(* Logix 5000 project; controller BTS01 vendor 1 type 14 code 217 rev 32.14; software revision 32.04 *)

TASK MainTask (continuous, watchdog 500 ms) : MainProgram, Alarm, CIP

MODULES
   Local : vendor 1 type 14 code 217 (5069 0, rev 32.14)
      Flow_Meter_01 : Promag_300_500 (Ethernet 10.10.1.3, rev 1.1, StandardDataDriven RPI 20 ms)
      FLEX5000 : 5094-AENTR (Ethernet 10.10.1.2, rev 4.1)
          : 5094-IF8 (5094 1, rev 2.1, StandardDataDriven RPI 100 ms)
          : 5094-OB16 (5094 5, rev 2.1, StandardDataDriven RPI 5 ms)
              FLEX5000:5:O.Pt09.Data   // RED STOP
              FLEX5000:5:O.Pt08.Data   // GREEN RUN
          : 5094-IB16 (5094 3, rev 2.1, StandardDataDriven RPI 5 ms)
          : 5094-IB16 (5094 6, rev 2.1, StandardDataDriven RPI 5 ms)
          : 5094-OF8 (5094 2, rev 2.1, StandardDataDriven RPI 100 ms)
          : 5094-OB16 (5094 4, rev 2.1, StandardDataDriven RPI 5 ms)
              FLEX5000:4:O.Pt13.Data   // Red
END_MODULES

TYPE CIP_PROGRAM :   // 30 STEP CIP PROGRAM
STRUCT
   NAME : STRING;   // CIP PROGRAM NAME
   NUMBER : INT;   // CIP PROGRAM NUMBER
   STEPS : CIP_STEP_DEF[50];   // CIP PROGRAM STEPS
END_STRUCT
END_TYPE

TYPE CIP_Recipe :
STRUCT
   Recipe_Name : STRING;
   Recipe_Description : STRING;
   Step_Desc : STRING[50];
   Step_Time : REAL[50];
END_STRUCT
END_TYPE

TYPE CIP_STEP_DEF :   // CIP SEQUENCER STEP DEFFINITION
STRUCT
   NAME : STRING;   // CIP STEP NAME
   TYPE : INT;   // CIP STEP TYPE
   TIME_SPT : REAL;   // CIP STEP TIME
   RETURN_TEMP_SPT : REAL;   // CIP RETURN STEP TEMP
   REF_FILE : DINT;   // CIP STEP REFERENCE FILE
   RETURN_COND_SPT : REAL;   // CIP RETURN STEP CONDUCTIVITY
END_STRUCT
END_TYPE

TYPE DateTime :
STRUCT
   Year : DINT;
   Month : DINT;
   Day : DINT;
   Hour : DINT;
   Minute : DINT;
   Second : DINT;
   MicroSecond : DINT;
END_STRUCT
END_TYPE

TYPE STRING64 :
STRUCT
   LEN : DINT;
   DATA : SINT[64];
END_STRUCT
END_TYPE

ADD_ON_INSTRUCTION DTE_Air_Valve_v2   (* revision 2.0 *)
VAR_INPUT
   CMD : BOOL; {visible}
END_VAR
VAR_OUTPUT
   TON_OUT_ACC : DINT; {access Read Only, visible}
   TOFF_OUT_ACC : DINT; {access Read Only, visible}
   OUT : BOOL; {access Read Only, required}
END_VAR
VAR_INPUT
   FB_DES : BOOL;
   FB_ACT : BOOL;
   ACK : BOOL;
END_VAR
VAR_OUTPUT
   ALARME : BOOL; {access Read Only}
END_VAR
VAR_INPUT
   ALM_PRE : DINT := 7000;
   ALM_AUTO_RESET_PRE : DINT;
   TON_OUT_PRE : DINT; {required}
   TOFF_OUT_PRE : DINT; {required}
   P : BOOL; {required}   // Process Command
   C : BOOL; {required}   // CIP Command
   M : DINT;
        .1   // Auto On
        .2   // Force On
        .3   // Force Off
   desc_nom : DINT;
   equip_nom : DINT;
   nom : DINT;
   Allowed : BOOL;
END_VAR
VAR_IN_OUT
   Description : STRING; {required}
   PIDName : STRING; {required}
END_VAR
VAR_INPUT
   Auto_On_PB : BOOL; {required}   // Momentary PB
   Manual_On_PB : BOOL; {required}   // Momentary PB
   Manual_Off_PB : BOOL; {required}   // Momentary PB
   Status : DINT; {visible}
END_VAR
VAR_OUTPUT
   ITEMTAG : DINT; {access Read Only, visible}
END_VAR
VAR_INPUT
   MOA_Mode : DINT; {visible}
END_VAR
VAR
   INTERNAL_TIM_ALM : TIMER := (PRE := 7000);
   INTERNAL_TIM_AUTO_RESET : TIMER;
   OUT_OFF_MEM : BOOL;
   OUT_ON_MEM : BOOL;
   INTERNAL_TON_OUT : TIMER;
   INTERNAL_TOFF_OUT : TIMER;
   Desc : STRING;
   ValveName : STRING; {access None}
   DisplayName : STRING;
END_VAR

ROUTINE Logic   (* ladder *)
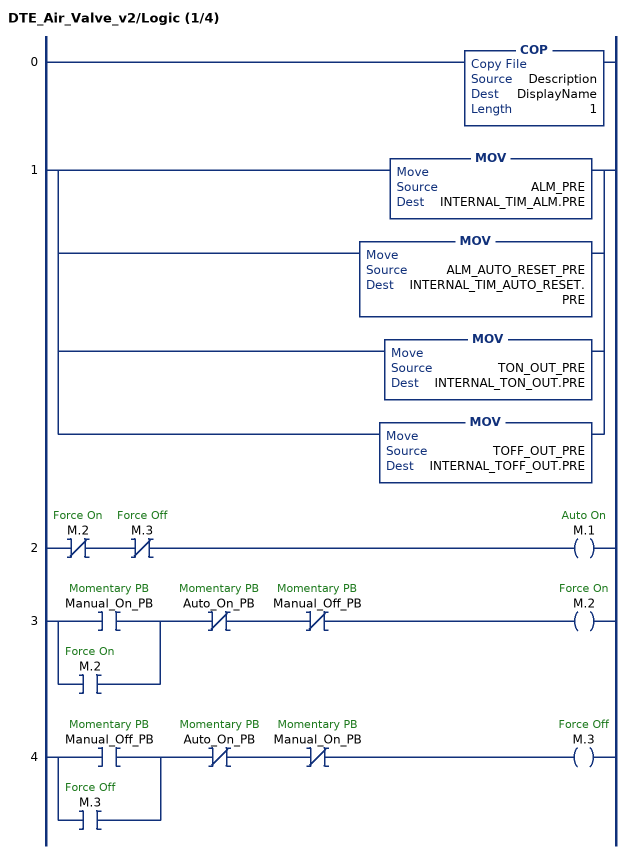
   0: COP(Description,DisplayName,1);
   1: [MOV(ALM_PRE,INTERNAL_TIM_ALM.PRE) ,MOV(ALM_AUTO_RESET_PRE,INTERNAL_TIM_AUTO_RESET.PRE) ,MOV(TON_OUT_PRE,INTERNAL_TON_OUT.PRE) ,MOV(TOFF_OUT_PRE,INTERNAL_TOFF_OUT.PRE) ];
   2: XIO(M.2)XIO(M.3)OTE(M.1);
   3: [XIC(Manual_On_PB) ,XIC(M.2) ]XIO(Auto_On_PB)XIO(Manual_Off_PB)OTE(M.2);
   4: [XIC(Manual_Off_PB) ,XIC(M.3) ]XIO(Auto_On_PB)XIO(Manual_On_PB)OTE(M.3);
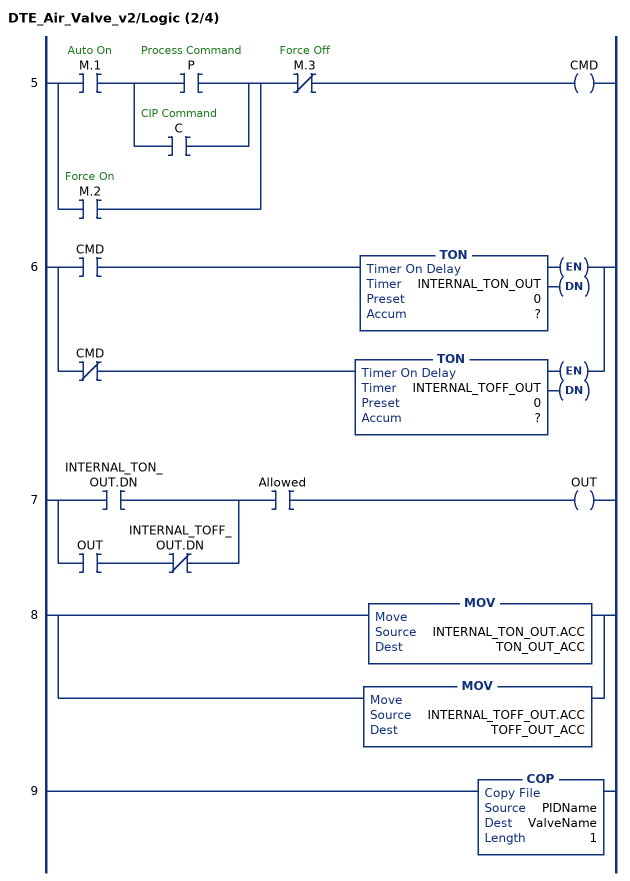
   5: [XIC(M.1) [XIC(P) ,XIC(C) ] ,XIC(M.2) ]XIO(M.3)OTE(CMD);
   6: [XIC(CMD) TON(INTERNAL_TON_OUT,?,?) ,XIO(CMD) TON(INTERNAL_TOFF_OUT,?,?) ];
   7: [XIC(INTERNAL_TON_OUT.DN) ,XIC(OUT) XIO(INTERNAL_TOFF_OUT.DN) ]XIC(Allowed)OTE(OUT);
   8: [MOV(INTERNAL_TON_OUT.ACC,TON_OUT_ACC) ,MOV(INTERNAL_TOFF_OUT.ACC,TOFF_OUT_ACC) ];
   9: COP(PIDName,ValveName,1);
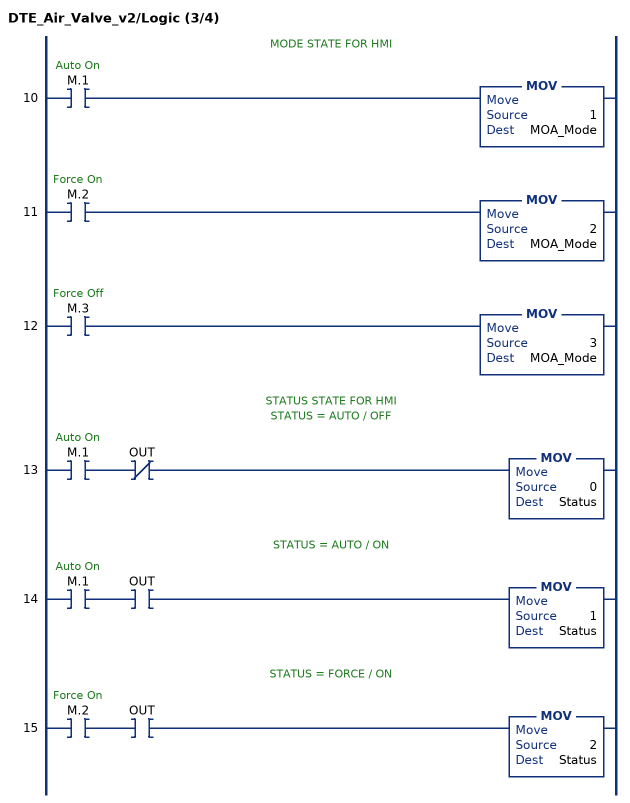
   // MODE STATE FOR HMI
   10: XIC(M.1)MOV(1,MOA_Mode);
   11: XIC(M.2)MOV(2,MOA_Mode);
   12: XIC(M.3)MOV(3,MOA_Mode);
   // STATUS STATE FOR HMI
   // STATUS = AUTO / OFF
   13: XIC(M.1)XIO(OUT)MOV(0,Status);
   // STATUS = AUTO / ON
   14: XIC(M.1)XIC(OUT)MOV(1,Status);
   // STATUS = FORCE / ON
   15: XIC(M.2)XIC(OUT)MOV(2,Status);
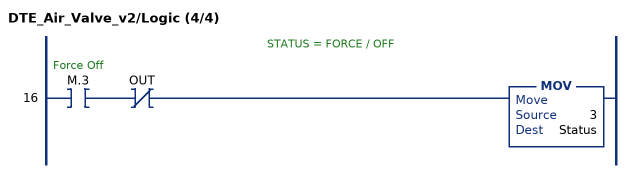
   // STATUS = FORCE / OFF
   16: XIC(M.3)XIO(OUT)MOV(3,Status);
END_ROUTINE
END_ADD_ON_INSTRUCTION

ADD_ON_INSTRUCTION DTE_MilliSec_TO_Min_Sec   (* revision 1.0, vendor DTE *)
// Convert Milliseconds to Minutes and Seconds
VAR_INPUT
   MSec_In_PRE : DINT; {required}   // PRE Milliseconds Input
   MSec_In_ACC : DINT; {access None, required}   // ACC Milliseconds Input
END_VAR
VAR_OUTPUT
   Sec_Out : DINT; {access Read Only, required}   // Seconds Output
   Min_Out : DINT; {access Read Only, required}   // Minutes Output
END_VAR
VAR_INPUT
   MSec_In : DINT;
END_VAR
VAR
   Sec_In_Conv : DINT; {access None}   // Seconds Input Converted From Milliseconds
END_VAR

ROUTINE Logic   (* ladder *)
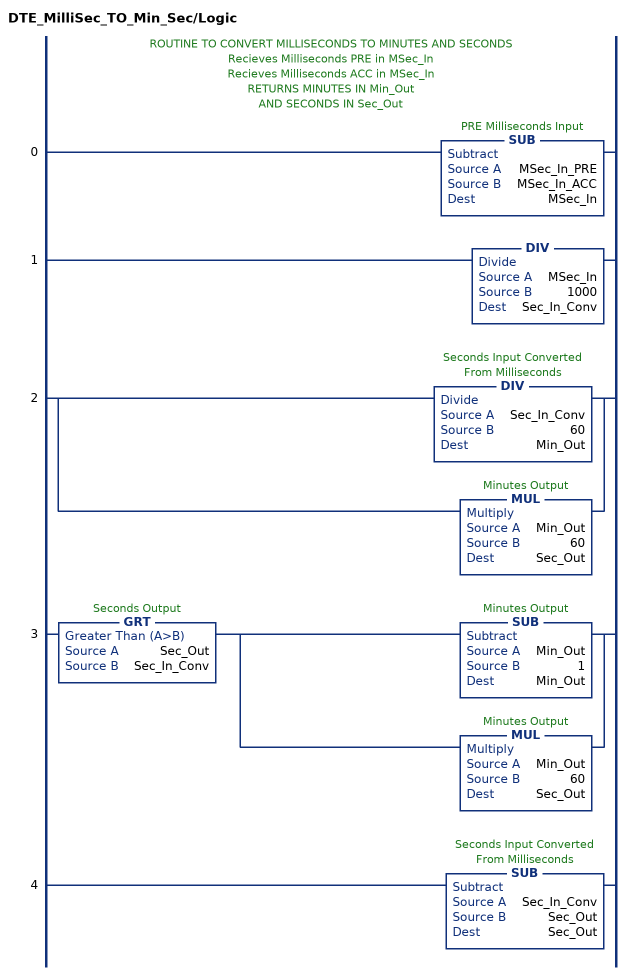
   // ROUTINE TO CONVERT MILLISECONDS TO MINUTES AND SECONDS
   // Recieves Milliseconds PRE in MSec_In
   // Recieves Milliseconds ACC in MSec_In
   // RETURNS MINUTES IN Min_Out
   // AND SECONDS IN Sec_Out
   0: SUB(MSec_In_PRE,MSec_In_ACC,MSec_In);
   1: DIV(MSec_In,1000,Sec_In_Conv);
   2: [DIV(Sec_In_Conv,60,Min_Out) ,MUL(Min_Out,60,Sec_Out) ];
   3: GRT(Sec_Out,Sec_In_Conv)[SUB(Min_Out,1,Min_Out) ,MUL(Min_Out,60,Sec_Out) ];
   4: SUB(Sec_In_Conv,Sec_Out,Sec_Out);
END_ROUTINE
END_ADD_ON_INSTRUCTION

ADD_ON_INSTRUCTION DTE_Motor_Starter_v2   (* revision 2.0, vendor DTE *)
// Revision note:
// Modified Interlock Logic
// Changed "Enable" to "Auto_Run_Enable"
VAR_INPUT
   AUTO_RUN_ENABLE : BOOL; {access None, required}   // SYSTEM RUN ENABLE IN AUTO MODE
   AUTO_PB : BOOL; {required}
   FORCE_ON_PB : BOOL; {required}
   FORCE_OFF_PB : BOOL; {required}
   JOG_PB : BOOL; {required}
   STARTER_AUX : BOOL; {required}   // RUN SIGNAL
   INTERLOCK : BOOL; {required}   // INTERLOCK IS ANY INPUT TO DISABLE THE STARTER
END_VAR
VAR_OUTPUT
   RUN_COMMAND : BOOL; {required}   // ENERGIZE STARTER
   STOPPED_WHILE_RUNNING : BOOL; {required}
   FAILED_TO_START : BOOL; {required}
   MOA_MODE : DINT; {access Read Only, required}
   STATUS : DINT; {access Read Only, required}
   ITEMTAG : DINT; {access Read Only, visible}
END_VAR
VAR
   Blink : TIMER := (PRE := 500); {access None}   // WILL BLINK THE LIGHT OUTPUT ON AND OFF FOR STATUS
   Blink_Unblink : TIMER := (PRE := 500); {access None}   // WILL UNBLINK THE LIGHT OUTPUT ON AND OFF FOR STATUS
   FAULT_DLY : TIMER := (PRE := 1500); {access None}   // THE MOTOR STARTER HAS THIS LONG TO ENERGIZE
   Motor_Has_Started_Timer : TIMER := (PRE := 1500); {access None}   // MOTOR STARTER AUX. INPUT HAS TO BE ON THIS LONG TO BE RUNNING
   MOTOR_HAS_RUN : BOOL; {access None}
   AUTO_MODE : BOOL;
   FORCE_ON_MODE : BOOL;
   FORCE_OFF_MODE : BOOL;
END_VAR

ROUTINE Logic   (* ladder *)
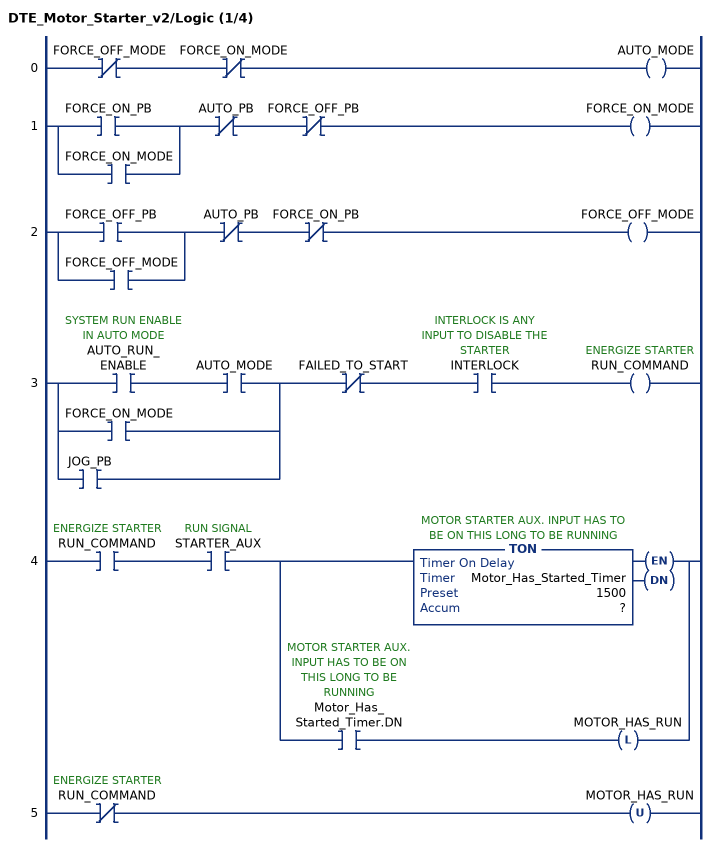
   0: XIO(FORCE_OFF_MODE)XIO(FORCE_ON_MODE)OTE(AUTO_MODE);
   1: [XIC(FORCE_ON_PB) ,XIC(FORCE_ON_MODE) ]XIO(AUTO_PB)XIO(FORCE_OFF_PB)OTE(FORCE_ON_MODE);
   2: [XIC(FORCE_OFF_PB) ,XIC(FORCE_OFF_MODE) ]XIO(AUTO_PB)XIO(FORCE_ON_PB)OTE(FORCE_OFF_MODE);
   3: [XIC(AUTO_RUN_ENABLE) XIC(AUTO_MODE) ,XIC(FORCE_ON_MODE) ,XIC(JOG_PB) ]XIO(FAILED_TO_START)XIC(INTERLOCK)OTE(RUN_COMMAND);
   4: XIC(RUN_COMMAND)XIC(STARTER_AUX)[TON(Motor_Has_Started_Timer,?,?) ,XIC(Motor_Has_Started_Timer.DN) OTL(MOTOR_HAS_RUN) ];
   5: XIO(RUN_COMMAND)OTU(MOTOR_HAS_RUN);
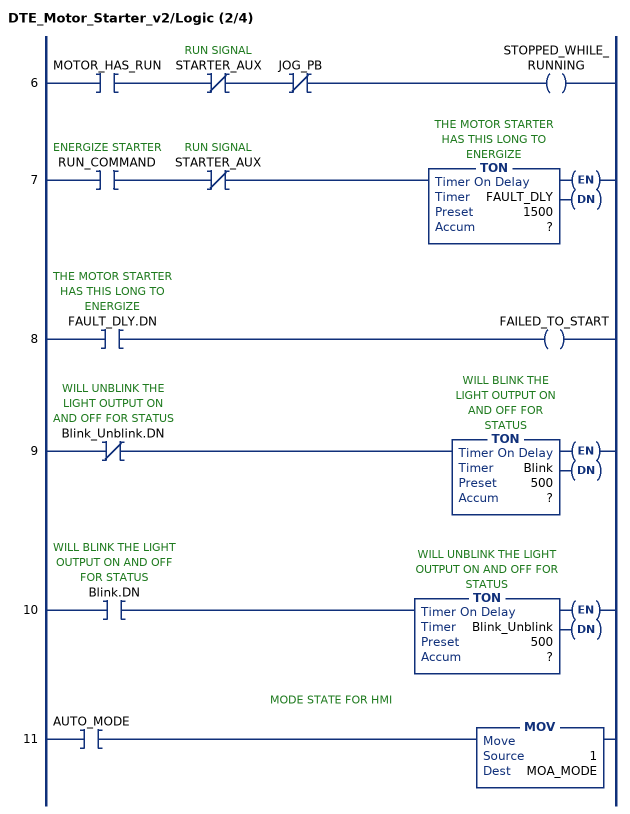
   6: XIC(MOTOR_HAS_RUN)XIO(STARTER_AUX)XIO(JOG_PB)OTE(STOPPED_WHILE_RUNNING);
   7: XIC(RUN_COMMAND)XIO(STARTER_AUX)TON(FAULT_DLY,?,?);
   8: XIC(FAULT_DLY.DN)OTE(FAILED_TO_START);
   9: XIO(Blink_Unblink.DN)TON(Blink,?,?);
   10: XIC(Blink.DN)TON(Blink_Unblink,?,?);
   // MODE STATE FOR HMI
   11: XIC(AUTO_MODE)MOV(1,MOA_MODE);
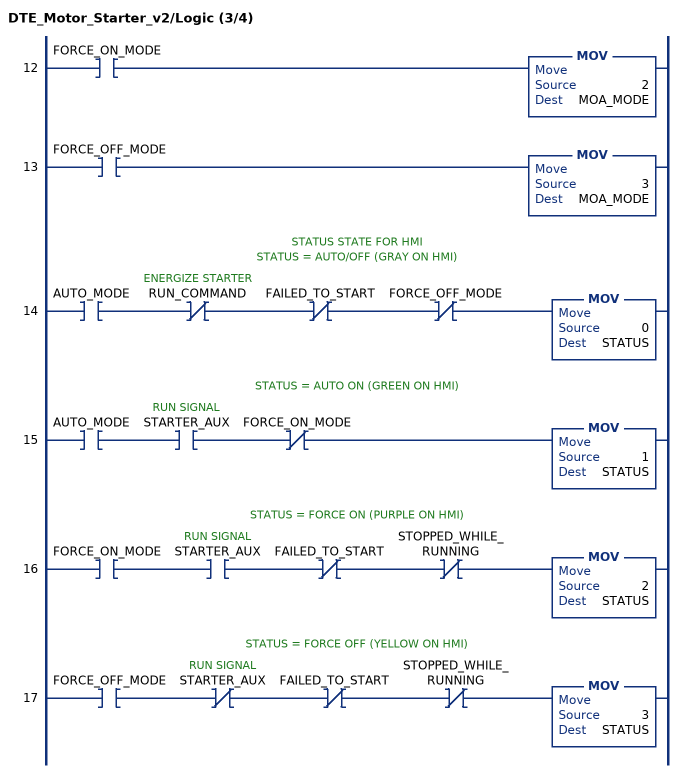
   12: XIC(FORCE_ON_MODE)MOV(2,MOA_MODE);
   13: XIC(FORCE_OFF_MODE)MOV(3,MOA_MODE);
   // STATUS STATE FOR HMI
   // STATUS = AUTO/OFF (GRAY ON HMI)
   14: XIC(AUTO_MODE)XIO(RUN_COMMAND)XIO(FAILED_TO_START)XIO(FORCE_OFF_MODE)MOV(0,STATUS);
   // STATUS = AUTO ON (GREEN ON HMI)
   15: XIC(AUTO_MODE)XIC(STARTER_AUX)XIO(FORCE_ON_MODE)MOV(1,STATUS);
   // STATUS = FORCE ON (PURPLE ON HMI)
   16: XIC(FORCE_ON_MODE)XIC(STARTER_AUX)XIO(FAILED_TO_START)XIO(STOPPED_WHILE_RUNNING)MOV(2,STATUS);
   // STATUS = FORCE OFF (YELLOW ON HMI)
   17: XIC(FORCE_OFF_MODE)XIO(STARTER_AUX)XIO(FAILED_TO_START)XIO(STOPPED_WHILE_RUNNING)MOV(3,STATUS);
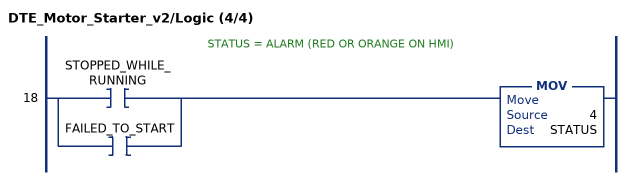
   // STATUS = ALARM (RED OR ORANGE ON HMI)
   18: [XIC(STOPPED_WHILE_RUNNING) ,XIC(FAILED_TO_START) ]MOV(4,STATUS);
END_ROUTINE
END_ADD_ON_INSTRUCTION

ADD_ON_INSTRUCTION DTE_SCP_W_LIM   (* revision 2.0, vendor Rockwell Automation Edited By DTE *)
// Scale w/Parameters
// with Min/Max Limit Control
// Help:
// Use this instruction to scale data from your analog module and bring it into the limits prescribed by the process variable or another analog module.
// Equations used in calculating a linear relationship:
// Scaled value = (input value - input min.) x rate + scaled minimum
// Rate = (scaled max. - scaled min.) / (input max. - input min.)
// Enabling the Limit_En Bit Limits the Output Value to the Scaled Min/Max Values. (09/16/16) DTK
VAR_INPUT
   Input : REAL; {required}
   Input_Min : REAL; {required}
   Input_Max : REAL; {required}
   Scaled_Min : REAL; {required}
   Scaled_Max : REAL; {required}
END_VAR
VAR_OUTPUT
   Output : REAL; {access Read Only, required}
END_VAR
VAR_INPUT
   Limit_En : BOOL; {visible}   // Limit Enable Bit Limits Output to Scaled Min/Max Values
END_VAR
VAR
   Rate : REAL;
END_VAR

ROUTINE Logic   (* ladder *)
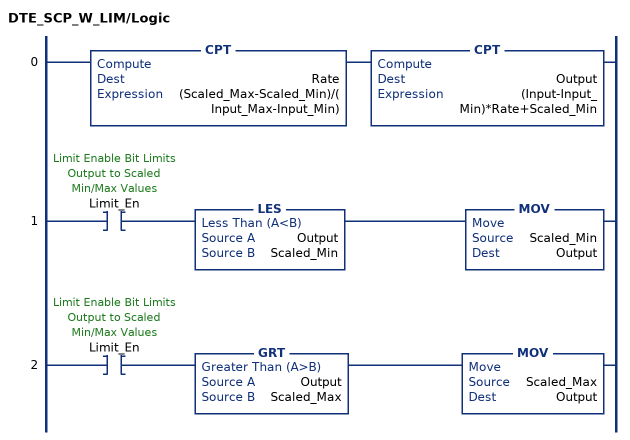
   0: CPT(Rate,(Scaled_Max-Scaled_Min)/(Input_Max-Input_Min))CPT(Output,(Input-Input_Min)*Rate+Scaled_Min);
   1: XIC(Limit_En)LES(Output,Scaled_Min)MOV(Scaled_Min,Output);
   2: XIC(Limit_En)GRT(Output,Scaled_Max)MOV(Scaled_Max,Output);
END_ROUTINE
END_ADD_ON_INSTRUCTION

ADD_ON_INSTRUCTION DTE_VFD   (* revision 2.0 2014_07_29, vendor DTE *)
// DeTroye Electric
// VFD Add-On Instruction
// Revision note:
// Removed Interlock from ForceOn Mode Logic
VAR_INPUT
   AUTO_PB : BOOL; {required}
   FORCE_ON_PB : BOOL; {required}
   FORCE_OFF_PB : BOOL; {required}
   REV_SELECT : BOOL;
   JOG_FWD_PB : BOOL;
   JOG_REV_PB : BOOL;
   AUTO_RUN_ENABLE : BOOL; {required}
   DRIVE_RUNNING : BOOL; {required}
   DRIVE_FAULTED : BOOL; {required}
   INTERLOCK : BOOL; {required}   // INTERLOCK IS ANY INPUT TO DISABLE THE DRIVE THERE IS NO DECEL EVERY OUTPUT GOES OFF ON LOSS OF THE INTERLOCK
   DISCONNECT_OFF : BOOL;
END_VAR
VAR_OUTPUT
   ENERGIZE_FWD_OUTPUT : BOOL; {access Read Only, required}
   ENERGIZE_REV_OUTPUT : BOOL; {access Read Only, visible}
   PILOT_LIGHT : BOOL; {visible}
END_VAR
VAR_INPUT
   SPEED_FWD : REAL; {required}
   SPEED_REV : REAL;
   AUTO_SPEED_SETPOINT : REAL; {required}
   FORCE_SPEED_SETPOINT : REAL; {required}
END_VAR
VAR_OUTPUT
   SPEED_0_TO_100_OUTPUT : REAL; {required}
END_VAR
VAR_INPUT
   SCALE_MIN_RAW : REAL; {access None}
   SCALED_MAX_RAW : REAL;
END_VAR
VAR_OUTPUT
   SPEED_REF_SCALED_RAW : REAL; {access Read Only}
   ITEMTAG : DINT; {access Read Only, visible}
END_VAR
VAR_INPUT
   MOA_MODE : DINT; {visible}
END_VAR
VAR_OUTPUT
   STATUS : DINT; {access Read Only, visible}
   DIRECTION_STATUS : DINT; {access Read Only}
END_VAR
VAR_INPUT
   VFD_ACCEL_TIME : DINT; {required}
END_VAR
VAR_OUTPUT
   STOPPED_WHILE_RUNNING : BOOL; {access Read Only, visible}
   FAILED_TO_START : BOOL; {access Read Only, visible}
END_VAR
VAR_INPUT
   Alarm_Ack : BOOL; {access Read Only, required}   // Acknowledge Alarm Input
END_VAR
VAR
   AUTO_RUN : BOOL; {access None}
   COMMANDED_SPEED : DINT; {access None}
   VFD_DTE : SCP; {access None}
   Blink_Fast : TIMER := (PRE := 250); {access None}
   Unblink_Fast : TIMER := (PRE := 250); {access None}
   AUTO_MODE : BOOL;
   FORCE_ON_MODE : BOOL;
   FORCE_OFF_MODE : BOOL;
   MOTOR_UP_TO_SPEED_TMR : TIMER := (PRE := 1500); {access None}
   VFD_RUNNING : BOOL; {access None}
   VFD_FAILED_TO_START_TMR : TIMER := (PRE := 1500); {access None}
   VFD_ACCEL_TIME_MULTIPLIER : DINT; {access None}
END_VAR

ROUTINE Logic   (* ladder *)
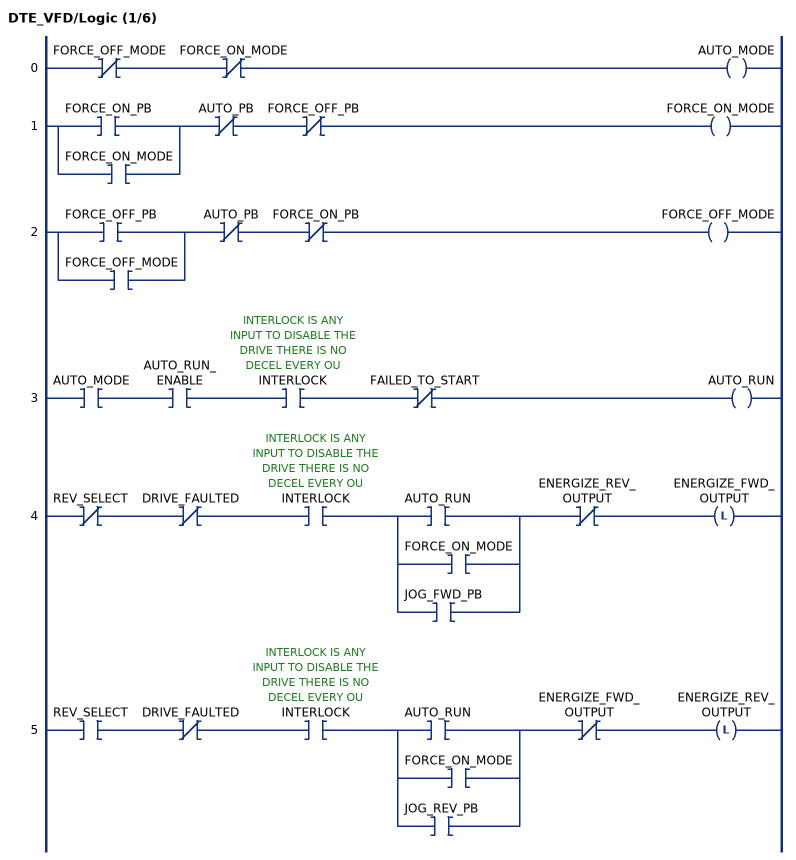
   0: XIO(FORCE_OFF_MODE)XIO(FORCE_ON_MODE)OTE(AUTO_MODE);
   1: [XIC(FORCE_ON_PB) ,XIC(FORCE_ON_MODE) ]XIO(AUTO_PB)XIO(FORCE_OFF_PB)OTE(FORCE_ON_MODE);
   2: [XIC(FORCE_OFF_PB) ,XIC(FORCE_OFF_MODE) ]XIO(AUTO_PB)XIO(FORCE_ON_PB)OTE(FORCE_OFF_MODE);
   3: XIC(AUTO_MODE)XIC(AUTO_RUN_ENABLE)XIC(INTERLOCK)XIO(FAILED_TO_START)OTE(AUTO_RUN);
   4: XIO(REV_SELECT)XIO(DRIVE_FAULTED)XIC(INTERLOCK)[XIC(AUTO_RUN) ,XIC(FORCE_ON_MODE) ,XIC(JOG_FWD_PB) ]XIO(ENERGIZE_REV_OUTPUT)OTL(ENERGIZE_FWD_OUTPUT);
   5: XIC(REV_SELECT)XIO(DRIVE_FAULTED)XIC(INTERLOCK)[XIC(AUTO_RUN) ,XIC(FORCE_ON_MODE) ,XIC(JOG_REV_PB) ]XIO(ENERGIZE_FWD_OUTPUT)OTL(ENERGIZE_REV_OUTPUT);
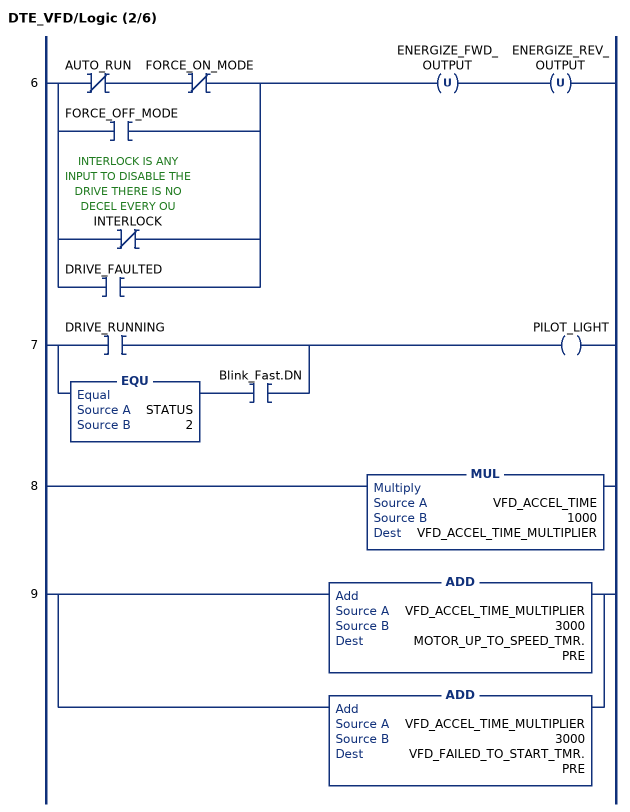
   6: [XIO(AUTO_RUN) XIO(FORCE_ON_MODE) ,XIC(FORCE_OFF_MODE) ,XIO(INTERLOCK) ,XIC(DRIVE_FAULTED) ]OTU(ENERGIZE_FWD_OUTPUT)OTU(ENERGIZE_REV_OUTPUT);
   7: [XIC(DRIVE_RUNNING) ,EQU(STATUS,2) XIC(Blink_Fast.DN) ]OTE(PILOT_LIGHT);
   8: MUL(VFD_ACCEL_TIME,1000,VFD_ACCEL_TIME_MULTIPLIER);
   9: [ADD(VFD_ACCEL_TIME_MULTIPLIER,3000,MOTOR_UP_TO_SPEED_TMR.PRE) ,ADD(VFD_ACCEL_TIME_MULTIPLIER,3000,VFD_FAILED_TO_START_TMR.PRE) ];
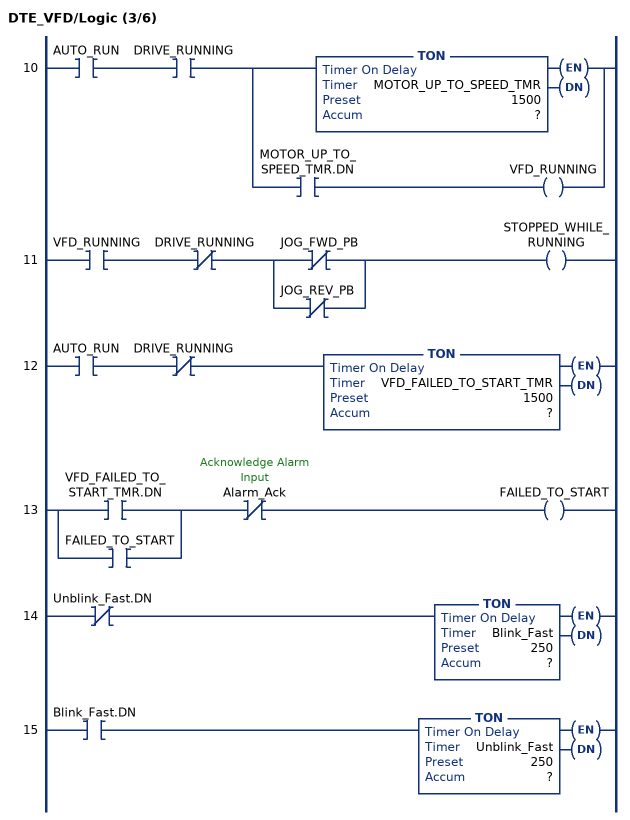
   10: XIC(AUTO_RUN)XIC(DRIVE_RUNNING)[TON(MOTOR_UP_TO_SPEED_TMR,?,?) ,XIC(MOTOR_UP_TO_SPEED_TMR.DN) OTE(VFD_RUNNING) ];
   11: XIC(VFD_RUNNING)XIO(DRIVE_RUNNING)[XIO(JOG_FWD_PB) ,XIO(JOG_REV_PB) ]OTE(STOPPED_WHILE_RUNNING);
   12: XIC(AUTO_RUN)XIO(DRIVE_RUNNING)TON(VFD_FAILED_TO_START_TMR,?,?);
   13: [XIC(VFD_FAILED_TO_START_TMR.DN) ,XIC(FAILED_TO_START) ]XIO(Alarm_Ack)OTE(FAILED_TO_START);
   14: XIO(Unblink_Fast.DN)TON(Blink_Fast,?,?);
   15: XIC(Blink_Fast.DN)TON(Unblink_Fast,?,?);
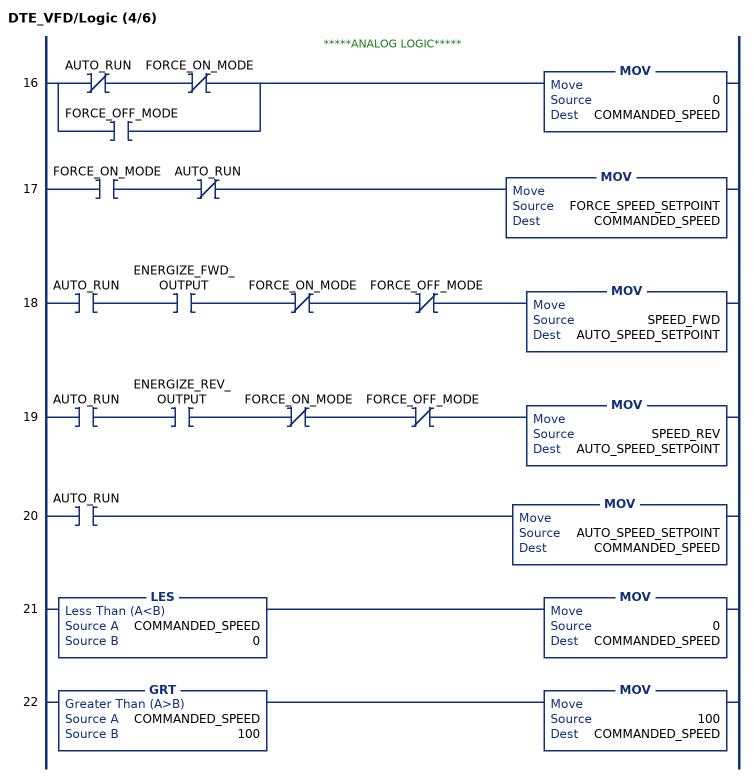
   // *****ANALOG LOGIC*****
   16: [XIO(AUTO_RUN) XIO(FORCE_ON_MODE) ,XIC(FORCE_OFF_MODE) ]MOV(0,COMMANDED_SPEED);
   17: XIC(FORCE_ON_MODE)XIO(AUTO_RUN)MOV(FORCE_SPEED_SETPOINT,COMMANDED_SPEED);
   18: XIC(AUTO_RUN)XIC(ENERGIZE_FWD_OUTPUT)XIO(FORCE_ON_MODE)XIO(FORCE_OFF_MODE)MOV(SPEED_FWD,AUTO_SPEED_SETPOINT);
   19: XIC(AUTO_RUN)XIC(ENERGIZE_REV_OUTPUT)XIO(FORCE_ON_MODE)XIO(FORCE_OFF_MODE)MOV(SPEED_REV,AUTO_SPEED_SETPOINT);
   20: XIC(AUTO_RUN)MOV(AUTO_SPEED_SETPOINT,COMMANDED_SPEED);
   21: LES(COMMANDED_SPEED,0)MOV(0,COMMANDED_SPEED);
   22: GRT(COMMANDED_SPEED,100)MOV(100,COMMANDED_SPEED);
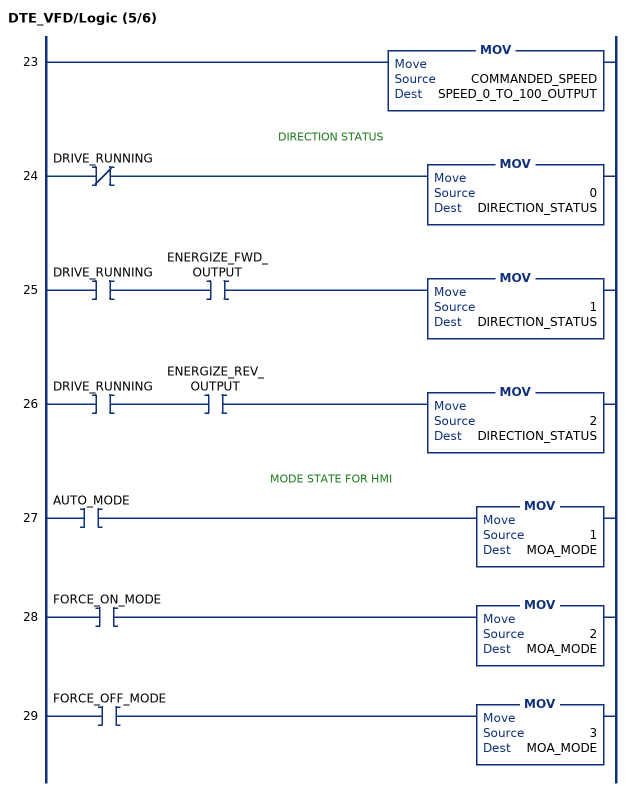
   23: MOV(COMMANDED_SPEED,SPEED_0_TO_100_OUTPUT);
   // DIRECTION STATUS
   24: XIO(DRIVE_RUNNING)MOV(0,DIRECTION_STATUS);
   25: XIC(DRIVE_RUNNING)XIC(ENERGIZE_FWD_OUTPUT)MOV(1,DIRECTION_STATUS);
   26: XIC(DRIVE_RUNNING)XIC(ENERGIZE_REV_OUTPUT)MOV(2,DIRECTION_STATUS);
   // MODE STATE FOR HMI
   27: XIC(AUTO_MODE)MOV(1,MOA_MODE);
   28: XIC(FORCE_ON_MODE)MOV(2,MOA_MODE);
   29: XIC(FORCE_OFF_MODE)MOV(3,MOA_MODE);
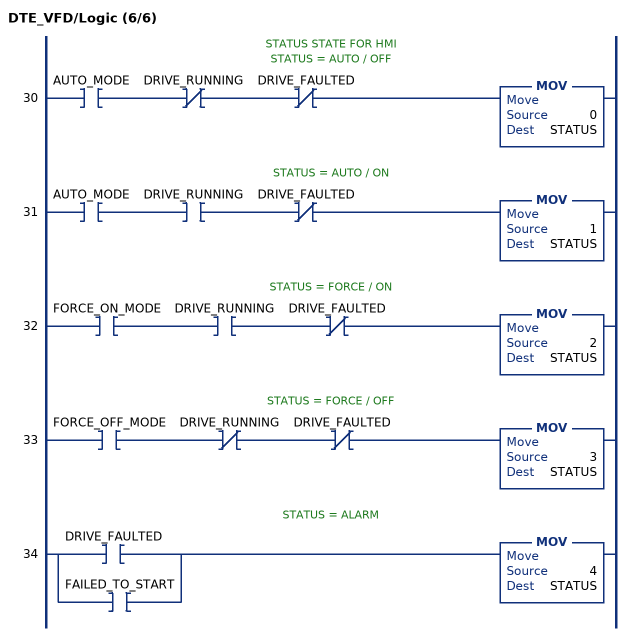
   // STATUS STATE FOR HMI
   // STATUS = AUTO / OFF
   30: XIC(AUTO_MODE)XIO(DRIVE_RUNNING)XIO(DRIVE_FAULTED)MOV(0,STATUS);
   // STATUS = AUTO / ON
   31: XIC(AUTO_MODE)XIC(DRIVE_RUNNING)XIO(DRIVE_FAULTED)MOV(1,STATUS);
   // STATUS = FORCE / ON
   32: XIC(FORCE_ON_MODE)XIC(DRIVE_RUNNING)XIO(DRIVE_FAULTED)MOV(2,STATUS);
   // STATUS = FORCE / OFF
   33: XIC(FORCE_OFF_MODE)XIO(DRIVE_RUNNING)XIO(DRIVE_FAULTED)MOV(3,STATUS);
   // STATUS = ALARM
   34: [XIC(DRIVE_FAULTED) ,XIC(FAILED_TO_START) ]MOV(4,STATUS);
END_ROUTINE
END_ADD_ON_INSTRUCTION

ADD_ON_INSTRUCTION Level_Sensor   (* revision 1.0 *)
VAR_INPUT
   RawInput : REAL; {required}   // Raw Input from Analog Input Card 0-30840
END_VAR
VAR_OUTPUT
   SensorPercentLevel : REAL; {access Read Only}   // Percent Level Before Additional Tank Parameters are Accounted for
   ActualPercentLevel : REAL; {access Read Only, required}   // Level in Percent
END_VAR
VAR_INPUT
   SensorUpperRange : REAL; {required}   // Scaled Upper Range of Sensor Set According to Sensor Name Plate or Programmed Upper Range Value
   TankOverFlow : REAL; {required}   // Inches from Sensor to Top of Over Flow
   TankCapacity : REAL; {required}   // Capacity of Tank in Gallons
   BelowSensor : REAL; {required}   // Gallons of Tank Capacity Below Sensor
   ProductDensity : REAL; {required}   // Product Density in lbs/gal
   Scaled_Min : REAL; {required}
   Scaled_Max : REAL; {required}
   Input_Min : REAL; {required}
   Input_Max : REAL; {required}
END_VAR
VAR_OUTPUT
   LBS : REAL; {access Read Only, visible}   // Lbs of Product in Tank
   KG : REAL; {access Read Only, visible}   // Kilograms of Product in Tank
END_VAR
VAR
   Offset : REAL;
   Slope : REAL;
   ProductDensity_lbs_per_Gal : REAL;
   SensorUpperRange_in : REAL;
   TankOverFlow_in : REAL;
   TankCapacity_gal : REAL;
   BelowSensor_gal : REAL;
END_VAR

ROUTINE Logic   (* ladder *)
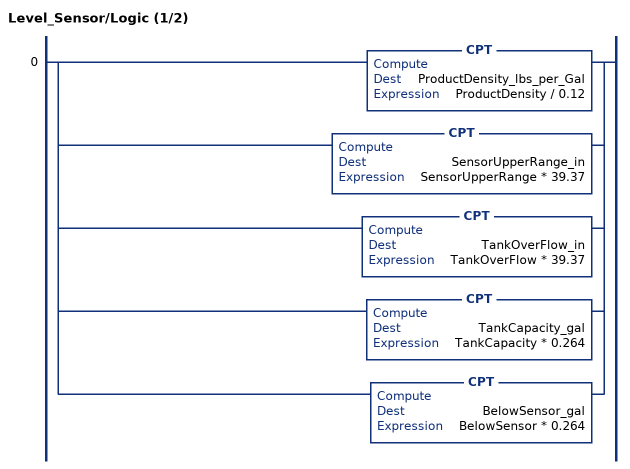
   0: [CPT(ProductDensity_lbs_per_Gal,ProductDensity / 0.12) ,CPT(SensorUpperRange_in,SensorUpperRange * 39.37) ,CPT(TankOverFlow_in,TankOverFlow * 39.37) ,CPT(TankCapacity_gal,TankCapacity * 0.264) ,CPT(BelowSensor_gal,BelowSensor * 0.264) ];
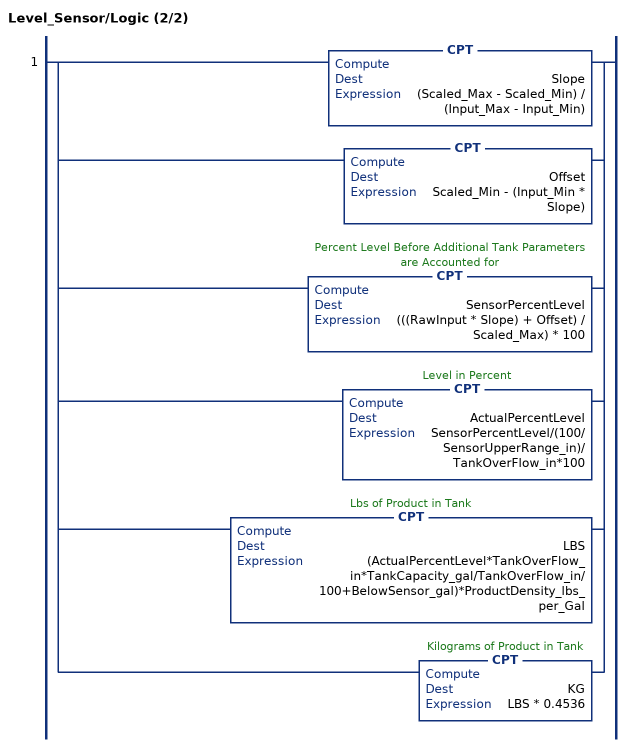
   1: [CPT(Slope,(Scaled_Max - Scaled_Min) / (Input_Max - Input_Min)) ,CPT(Offset,Scaled_Min - (Input_Min * Slope)) ,CPT(SensorPercentLevel,(((RawInput * Slope) + Offset) / Scaled_Max) * 100) ,CPT(ActualPercentLevel,SensorPercentLevel/(100/SensorUpperRange_in)/TankOverFlow_in*100) ,CPT(LBS,(ActualPercentLevel*TankOverFlow_in*TankCapacity_gal/TankOverFlow_in/100+BelowSensor_gal)*ProductDensity_lbs_per_Gal) ,CPT(KG,LBS * 0.4536) ];
END_ROUTINE
END_ADD_ON_INSTRUCTION
